TYPE ST_PosInterface :
STRUCT
	PosControl AT%Q* : POS_Control;
	PosStatus AT%I* : POS_Status;
	StmControl AT%Q* : STM_Control;
	StmStatus AT%I* : STM_Status;
END_STRUCT
END_TYPE

(* stored: Version 1.1.0.1, ProductVersion 3.1.4024.3
   DUT ST_PosInterface: Id {533b91df-859d-4fc2-aeae-dd3c796626c2} *)
